(* PLC project presence_sensor, Dassault Systèmes ControlBuild 2024x *)
(* stored: creationDateTime 2023-10-04T11:03:51-01:00 *)

(* This module simulates the behaviour of a presence sensor that detects products. *)
FUNCTION_BLOCK motion_lib.presence_sensor
  VAR_INPUT
    incPositionX : REAL := 0.0;
    incPositionY : REAL := 0.0;
    incPositionZ : REAL := 0.0;
  END_VAR
  VAR_INPUT
    coordCenterX : REAL := 0.0;
    coordCenterY : REAL := 0.0;
    coordCenterZ : REAL := 0.0;
    incRotationX : REAL := 0.0;
    incRotationY : REAL := 0.0;
    incRotationZ : REAL := 0.0;
  END_VAR
  VAR_INPUT
    sensorSupply : BOOL := true;
  END_VAR
  VAR_OUTPUT
    presence : BOOL := false;
  END_VAR
  VAR
    status_act_prod : DINT := 0;
    m11 : REAL := 1.0;
    m12 : REAL := 0.0;
    m13 : REAL := 0.0;
    m14 : REAL := 0.0;
    m21 : REAL := 0.0;
    m22 : REAL := 1.0;
    m23 : REAL := 0.0;
    m24 : REAL := 0.0;
    m31 : REAL := 0.0;
    m32 : REAL := 0.0;
    m33 : REAL := 1.0;
    m34 : REAL := 0.0;
    m41 : REAL := 0.0;
    m42 : REAL := 0.0;
    m43 : REAL := 0.0;
    m44 : REAL := 1.0;
    detection : BOOL := false;
  END_VAR
  VAR CONSTANT
    presenceLogic : BOOL := true;
  END_VAR
  VAR
    d_presence : BOOL := false;
    v_d_presence : BOOL := true;
  END_VAR


ACTION C_source_code:
/* ----------------------------------------------------------------	*/
/* Type : Model of Operative Behaviour					*/
/* Category :  Actors and Products						*/
/* Author : Dassault Systemes						*/
/* Update date : June 2018							*/
/* ----------------------------------------------------------------	*/
/* This module simulates the behaviour of a presence sensor that 	*/
/* detects products.								*/
/* It is an "actor" and can be shifted or rotated.			*/
/* The product that is in interaction should modify the variable 	*/
/* "detection".								*/
/* ----------------------------------------------------------------	*/


/* Management of the detection	*/
if (d_presence) presence = v_d_presence;
else 
	presence = sensorSupply & (detection ^ ! presenceLogic);


/* Reset informations given by the product	*/
detection = 0;

/* Association with a traverser : take account of the traverse speed	*/
if ((incPositionX != 0.0) || (incPositionY != 0.0) || (incPositionZ != 0.0))
	moveBy(myself, incPositionX, incPositionY, incPositionZ);

/* Association with a rotary plate ring : take account of the rotation speed	*/
if ((incRotationX != 0.0) || (incRotationY != 0.0) || (incRotationZ != 0.0))
	rotateBy(myself, incRotationX, incRotationY, incRotationZ, coordCenterX, coordCenterY, coordCenterZ);
END_ACTION
END_FUNCTION_BLOCK
